TYPE "Peeler_Status"
VERSION : 0.1
// Block: Peeler_Status
   STRUCT
      Lift : ValveMachine_COut;
      Extension : ValveMachine_COut;
      Is_Up : Bool;
      Is_Dwn : Bool;
   END_STRUCT;

END_TYPE
